// TIA Portal V18 export
VAR_GLOBAL   // PLC tag table "Cabinet_3"
   Sz3_Button_LED_ST29_ST30 AT %Q1300.0 : Bool;
   Sz3_Button_LED_ST30_ST31 AT %Q1300.1 : Bool;
   Sz3_Button_LED_ST18_ST37 AT %Q1300.2 : Bool;
   Sz3_Button_LED_ST19_ST18 AT %Q1300.3 : Bool;
   Sz3_Button_LED_ST20_ST19 AT %Q1300.4 : Bool;
   Sz3_Button_LED_Centering_ST19 AT %Q1300.5 : Bool;
   Sz3_Button_LED_Centering_ST18 AT %Q1300.6 : Bool;
   "Reserved(43)" AT %Q1300.7 : Bool;
   Sz3_ST29_SenA AT %I1300.0 : Bool;
   Sz3_ST29_SenB AT %I1300.1 : Bool;
   Sz3_ST29_SenC AT %I1300.2 : Bool;
   Sz3_ST29_SenD AT %I1300.3 : Bool;
   Sz3_ST30_SenA AT %I1300.4 : Bool;
   Sz3_ST30_SenB AT %I1300.5 : Bool;
   Sz3_ST30_SenC AT %I1300.6 : Bool;
   Sz3_ST30_SenD AT %I1300.7 : Bool;
   Sz3_ST31_SenA AT %I1301.0 : Bool;
   Sz3_ST31_SenB AT %I1301.1 : Bool;
   Sz3_ST31_SenC AT %I1301.2 : Bool;
   Sz3_ST31_SenD AT %I1301.3 : Bool;
   Sz3_ST18_SenA AT %I1301.4 : Bool;
   Sz3_ST18_SenB AT %I1301.5 : Bool;
   Sz3_ST18_SenC AT %I1301.6 : Bool;
   Sz3_ST18_SenD AT %I1301.7 : Bool;
   Sz3_ST19_SenA AT %I1302.0 : Bool;
   Sz3_ST19_SenB AT %I1302.1 : Bool;
   Sz3_ST19_SenC AT %I1302.2 : Bool;
   Sz3_ST19_SenD AT %I1302.3 : Bool;
   Sz3_ST20_SenA AT %I1302.4 : Bool;
   Sz3_ST20_SenB AT %I1302.5 : Bool;
   Sz3_ST20_SenC AT %I1302.6 : Bool;
   Sz3_ST20_SenD AT %I1302.7 : Bool;
   Sz3_Button_ST29_ST30 AT %I1303.0 : Bool;
   Sz3_Button_ST30_ST31 AT %I1303.1 : Bool;
   Sz3_Button_ST31_ST32 AT %I1303.2 : Bool;
   Sz3_Button_ST18_ST37 AT %I1303.3 : Bool;
   Sz3_Button_ST19_ST18 AT %I1303.4 : Bool;
   Sz3_Button_ST20_ST19 AT %I1303.5 : Bool;
   Sz3_Button_Centering_ST19 AT %I1303.6 : Bool;
   Sz3_Button_Centering_ST18 AT %I1303.7 : Bool;
   Sz3_Safety1_1 AT %I1304.0 : Bool;
   "Reserved(44)" AT %I1304.1 : Bool;
   "Reserved(45)" AT %I1304.2 : Bool;
   "Reserved(46)" AT %I1304.3 : Bool;
   Sz3_Safety1_2 AT %I1304.4 : Bool;
   "Reserved(47)" AT %I1304.5 : Bool;
   "Reserved(48)" AT %I1304.6 : Bool;
   "Reserved(49)" AT %I1304.7 : Bool;
   "Reserved(50)" AT %I1305.0 : Bool;
   "Reserved(51)" AT %I1305.1 : Bool;
   "Reserved(52)" AT %I1305.2 : Bool;
   "Reserved(53)" AT %I1305.3 : Bool;
   "Reserved(54)" AT %I1305.4 : Bool;
   "Reserved(55)" AT %I1305.5 : Bool;
   "Reserved(56)" AT %I1305.6 : Bool;
   "Reserved(57)" AT %I1305.7 : Bool;
END_VAR
